(* CoDeSys 2.3 library: WagoLibDaylightSaving.lib *)

(* POU SysRtcGetDS, ST *)
FUNCTION SysRtcGetDS : BOOL
VAR_INPUT
	dummy: BOOL;
END_VAR
VAR
END_VAR
;
END_FUNCTION

(* POU SysRtcSetDS, ST *)
FUNCTION SysRtcSetDS : BOOL
VAR_INPUT
	DaylightSaving: BOOL;
END_VAR
VAR
END_VAR
;
END_FUNCTION
